TYPE E_TankState :
(
    IDLE     := 0,
    FILLING  := 1,
    FULL     := 2,
    DRAINING := 3,
    FAULT    := 99
);
END_TYPE

(* stored: Version 1.1.0.1, ProductVersion 3.1.4024.16
   DUT E_TankState: Id {55881385-7f50-4a97-a637-fb03b40f86d4} *)
